{attribute 'pack_mode' := '1'}
TYPE ST_RemoveStationDataIn :
STRUCT
	sCellID						: STRING(30);
	sStationID					: STRING(30);
END_STRUCT
END_TYPE

(* stored: Version 1.1.0.1, ProductVersion 3.1.4024.5
   DUT ST_RemoveStationDataIn: Id {deef2b39-4b54-422b-a66e-387c7b5e724a} *)
